KUKA KRL data list: Mein_Job.dat

&ACCESS RVP
&PARAM EDITMASK = *
DEFDAT  Mein_Job
;FOLD EXTERNAL DECLARATIONS;%{PE}%MKUKATPBASIS,%CEXT,%VCOMMON,%P
;FOLD BASISTECH EXT;%{PE}%MKUKATPBASIS,%CEXT,%VEXT,%P
EXT  BAS (BAS_COMMAND  :IN,REAL  :IN )
DECL INT SUCCESS
;ENDFOLD (BASISTECH EXT)
;FOLD USER EXT;%{E}%MKUKATPUSER,%CEXT,%VEXT,%P
;Make your modifications here

;ENDFOLD (USER EXT)
;ENDFOLD (EXTERNAL DECLARATIONS)

INT APP_GENNUMBER = 696359
INT APP_ANSWER
INT APP_OFFSET
DECL STATE_T APP_STATE


DECL PDAT PPDATP3={VEL 100,ACC 100,APO_DIST 100,GEAR_JERK 50.0000}
DECL FDAT FP15={TOOL_NO 0,BASE_NO 0,IPO_FRAME #BASE,POINT2[] " ",TQ_STATE FALSE}
DECL E6POS XP15={X 427.4689,Y 0,Z 804.78462,A 180,B -11.62509,C 180,S 2,T 2,E1 0,E2 0,E3 0,E4 0,E5 0,E6 0}
DECL PDAT PPDATP1={VEL 100,ACC 100,APO_DIST 100,GEAR_JERK 50.0000}
DECL FDAT FP1={TOOL_NO 0,BASE_NO 0,IPO_FRAME #BASE,POINT2[] " ",TQ_STATE FALSE}
DECL E6POS XP1={X -301.66101,Y -302.8701,Z 804.78462,A 45.11459,B -11.62509,C 180,S 2,T 2,E1 0,E2 0,E3 0,E4 0,E5 0,E6 0}
DECL LDAT LCPDATP15={VEL 1,ACC 100,APO_DIST 100,APO_FAC 50.0,ORI_TYP #VAR,CIRC_TYP #BASE,JERK_FAC 50.0}
DECL FDAT FP17={TOOL_NO 1,BASE_NO 0,IPO_FRAME #BASE,POINT2[] " ",TQ_STATE FALSE}
DECL E6POS XP17={X -347.18723,Y -317.7877,Z 219.17578,A -103.07185,B 84.54091,C 90.0003,S 2,T 34,E1 0,E2 0,E3 0,E4 0,E5 0,E6 0}
DECL LDAT LCPDATP1={VEL 1,ACC 100,APO_DIST 100,APO_FAC 50.0,ORI_TYP #VAR,CIRC_TYP #BASE,JERK_FAC 50.0}
DECL FDAT FP2={TOOL_NO 1,BASE_NO 0,IPO_FRAME #BASE,POINT2[] " ",TQ_STATE FALSE}
DECL E6POS XP2={X -382.02608,Y -317.7877,Z 206.99982,A -103.07185,B 84.54091,C 90.0003,S 2,T 34,E1 0,E2 0,E3 0,E4 0,E5 0,E6 0}
DECL LDAT LCPDATP2={VEL 1,ACC 100,APO_DIST 100,APO_FAC 50.0,ORI_TYP #VAR,CIRC_TYP #BASE,JERK_FAC 50.0}
DECL FDAT FP3={TOOL_NO 1,BASE_NO 0,IPO_FRAME #BASE,POINT2[] " ",TQ_STATE FALSE}
DECL E6POS XP3={X -387.87999,Y -342.9989,Z 206.99983,A -133.07183,B 84.54092,C 90.00032,S 2,T 34,E1 0,E2 0,E3 0,E4 0,E5 0,E6 0}
DECL LDAT LCPDATP3={VEL 1,ACC 100,APO_DIST 100,APO_FAC 50.0,ORI_TYP #VAR,CIRC_TYP #BASE,JERK_FAC 50.0}
DECL FDAT FP4={TOOL_NO 1,BASE_NO 0,IPO_FRAME #BASE,POINT2[] " ",TQ_STATE FALSE}
DECL E6POS XP4={X -405.55523,Y -361.90549,Z 206.99983,A -163.07189,B 84.54094,C 90.00025,S 2,T 2,E1 0,E2 0,E3 0,E4 0,E5 0,E6 0}
DECL LDAT LCPDATP4={VEL 1,ACC 100,APO_DIST 100,APO_FAC 50.0,ORI_TYP #VAR,CIRC_TYP #BASE,JERK_FAC 50.0}
DECL FDAT FP5={TOOL_NO 1,BASE_NO 0,IPO_FRAME #BASE,POINT2[] " ",TQ_STATE FALSE}
DECL E6POS XP5={X -430.31573,Y -369.44145,Z 206.99982,A 166.92797,B 84.54095,C 90.00012,S 2,T 2,E1 0,E2 0,E3 0,E4 0,E5 0,E6 0}
DECL LDAT LCPDATP5={VEL 1,ACC 100,APO_DIST 100,APO_FAC 50.0,ORI_TYP #VAR,CIRC_TYP #BASE,JERK_FAC 50.0}
DECL FDAT FP6={TOOL_NO 1,BASE_NO 0,IPO_FRAME #BASE,POINT2[] " ",TQ_STATE FALSE}
DECL E6POS XP6={X -455.52693,Y -363.58754,Z 206.99981,A 136.92781,B 84.54095,C 89.99995,S 2,T 2,E1 0,E2 0,E3 0,E4 0,E5 0,E6 0}
DECL LDAT LCPDATP6={VEL 1,ACC 100,APO_DIST 100,APO_FAC 50.0,ORI_TYP #VAR,CIRC_TYP #BASE,JERK_FAC 50.0}
DECL FDAT FP7={TOOL_NO 1,BASE_NO 0,IPO_FRAME #BASE,POINT2[] " ",TQ_STATE FALSE}
DECL E6POS XP7={X -474.43352,Y -345.91231,Z 206.99979,A 106.92766,B 84.54094,C 89.9998,S 2,T 42,E1 0,E2 0,E3 0,E4 0,E5 0,E6 0}
DECL LDAT LCPDATP7={VEL 1,ACC 100,APO_DIST 100,APO_FAC 50.0,ORI_TYP #VAR,CIRC_TYP #BASE,JERK_FAC 50.0}
DECL FDAT FP8={TOOL_NO 1,BASE_NO 0,IPO_FRAME #BASE,POINT2[] " ",TQ_STATE FALSE}
DECL E6POS XP8={X -481.96948,Y -321.15181,Z 206.99978,A 76.92756,B 84.54093,C 89.9997,S 2,T 42,E1 0,E2 0,E3 0,E4 0,E5 0,E6 0}
DECL LDAT LCPDATP8={VEL 1,ACC 100,APO_DIST 100,APO_FAC 50.0,ORI_TYP #VAR,CIRC_TYP #BASE,JERK_FAC 50.0}
DECL FDAT FP9={TOOL_NO 1,BASE_NO 0,IPO_FRAME #BASE,POINT2[] " ",TQ_STATE FALSE}
DECL E6POS XP9={X -476.11557,Y -295.94061,Z 206.99978,A 46.92754,B 84.54091,C 89.99968,S 2,T 42,E1 0,E2 0,E3 0,E4 0,E5 0,E6 0}
DECL LDAT LCPDATP9={VEL 1,ACC 100,APO_DIST 100,APO_FAC 50.0,ORI_TYP #VAR,CIRC_TYP #BASE,JERK_FAC 50.0}
DECL FDAT FP10={TOOL_NO 1,BASE_NO 0,IPO_FRAME #BASE,POINT2[] " ",TQ_STATE FALSE}
DECL E6POS XP10={X -458.44033,Y -277.03402,Z 206.99978,A 16.92761,B 84.5409,C 89.99975,S 2,T 42,E1 0,E2 0,E3 0,E4 0,E5 0,E6 0}
DECL LDAT LCPDATP10={VEL 1,ACC 100,APO_DIST 100,APO_FAC 50.0,ORI_TYP #VAR,CIRC_TYP #BASE,JERK_FAC 50.0}
DECL FDAT FP11={TOOL_NO 1,BASE_NO 0,IPO_FRAME #BASE,POINT2[] " ",TQ_STATE FALSE}
DECL E6POS XP11={X -433.67984,Y -269.49806,Z 206.99979,A -13.07226,B 84.54089,C 89.99988,S 2,T 42,E1 0,E2 0,E3 0,E4 0,E5 0,E6 0}
DECL LDAT LCPDATP11={VEL 1,ACC 100,APO_DIST 100,APO_FAC 50.0,ORI_TYP #VAR,CIRC_TYP #BASE,JERK_FAC 50.0}
DECL FDAT FP12={TOOL_NO 1,BASE_NO 0,IPO_FRAME #BASE,POINT2[] " ",TQ_STATE FALSE}
DECL E6POS XP12={X -408.46863,Y -275.35197,Z 206.9998,A -43.0721,B 84.54089,C 90.00005,S 2,T 42,E1 0,E2 0,E3 0,E4 0,E5 0,E6 0}
DECL LDAT LCPDATP12={VEL 1,ACC 100,APO_DIST 100,APO_FAC 50.0,ORI_TYP #VAR,CIRC_TYP #BASE,JERK_FAC 50.0}
DECL FDAT FP13={TOOL_NO 1,BASE_NO 0,IPO_FRAME #BASE,POINT2[] " ",TQ_STATE FALSE}
DECL E6POS XP13={X -389.56205,Y -293.0272,Z 206.99981,A -73.07194,B 84.54089,C 90.0002,S 2,T 34,E1 0,E2 0,E3 0,E4 0,E5 0,E6 0}
DECL LDAT LCPDATP13={VEL 1,ACC 100,APO_DIST 100,APO_FAC 50.0,ORI_TYP #VAR,CIRC_TYP #BASE,JERK_FAC 50.0}
DECL FDAT FP14={TOOL_NO 1,BASE_NO 0,IPO_FRAME #BASE,POINT2[] " ",TQ_STATE FALSE}
DECL E6POS XP14={X -382.02608,Y -317.7877,Z 206.99982,A -73.07194,B 84.54089,C 90.0002,S 2,T 34,E1 0,E2 0,E3 0,E4 0,E5 0,E6 0}
DECL LDAT LCPDATP16={VEL 1,ACC 100,APO_DIST 100,APO_FAC 50.0,ORI_TYP #VAR,CIRC_TYP #BASE,JERK_FAC 50.0}
DECL FDAT FP18={TOOL_NO 1,BASE_NO 0,IPO_FRAME #BASE,POINT2[] " ",TQ_STATE FALSE}
DECL E6POS XP18={X -364.111,Y -317.7877,Z 221.15063,A -73.07194,B 84.54089,C 90.0002,S 2,T 34,E1 0,E2 0,E3 0,E4 0,E5 0,E6 0}
DECL LDAT LCPDATP14={VEL 1,ACC 100,APO_DIST 100,APO_FAC 50.0,ORI_TYP #VAR,CIRC_TYP #BASE,JERK_FAC 50.0}
DECL FDAT FP16={TOOL_NO 1,BASE_NO 0,IPO_FRAME #BASE,POINT2[] " ",TQ_STATE FALSE}
DECL E6POS XP16={X -267.15455,Y -317.7877,Z 398.95974,A -73.07194,B 84.54089,C 90.0002,S 2,T 34,E1 0,E2 0,E3 0,E4 0,E5 0,E6 0}

ENDDAT
